// TIA Portal V15.1 export
// export: Created 2024-06-21T08:41:21.2470041Z, ExportSetting WithDefaults, DisplayName Totally Integrated Automation Portal, DisplayVersion V15.1 Update 5, DisplayName TIA Portal Openness, DisplayVersion V15.1 Update 5, DisplayName SINAMICS Startdrive Advanced, DisplayVersion V15.1, DisplayName G130, G150, S120, S150, SINAMICS MV, S210, DisplayVersion V15.1, DisplayName G110M, G120, G120C, G120D, G120P, DisplayVersion V15.1, DisplayName STEP 7 Professional, DisplayVersion V15.1 Update 5, DisplayName STEP 7 Safety, DisplayVersion V15.1, DisplayName WinCC Professional, DisplayVersion V15.1 Update 5, DisplayName SIMATIC Visualization Architect, DisplayVersion V15.1
FUNCTION_BLOCK "LVIDSQualityRequest"   // FB1220, SCL
{ S7_Optimized_Access := 'TRUE' }
VERSION : 0.1
// stored: AutoNumber false, IsIECCheckEnabled false, IsRetainMemResEnabled false, MemoryReserve 100, SetENOAutomatically False, UDAEnableTagReadback false
   VAR_INPUT
      I_TagID { ExternalAccessible := 'False'; ExternalVisible := 'False'; ExternalWritable := 'False'} : DWord;   // Tag ID
      I_BodyID { ExternalAccessible := 'False'; ExternalVisible := 'False'; ExternalWritable := 'False'} : DWord;   // Body ID
      I_CarrierID { ExternalAccessible := 'False'; ExternalVisible := 'False'; ExternalWritable := 'False'} : DWord;   // Carrier ID
      I_MixNr { ExternalAccessible := 'False'; ExternalVisible := 'False'; ExternalWritable := 'False'} : DWord;   // Mix Nr
      I_PopID { ExternalAccessible := 'False'; ExternalVisible := 'False'; ExternalWritable := 'False'} : UDInt;   // Spare Data / PopID
      I_PopIDSuffix { ExternalAccessible := 'False'; ExternalVisible := 'False'; ExternalWritable := 'False'} : Char;   // PopID suffix
      I_PopType { ExternalAccessible := 'False'; ExternalVisible := 'False'; ExternalWritable := 'False'} : UDInt;   // Pop identifier
      I_ManualModeVisible { ExternalAccessible := 'False'; ExternalVisible := 'False'; ExternalWritable := 'False'} : Bool := 0;   // 0= Hidden 1= Visible
      I_Start { ExternalAccessible := 'False'; ExternalVisible := 'False'; ExternalWritable := 'False'} : Bool;   // Start command
   END_VAR
   VAR_OUTPUT
      O_DataModeAuto { ExternalAccessible := 'False'; ExternalVisible := 'False'; ExternalWritable := 'False'} : Bool;   // Data mode - Automatic
      O_DataModeMan { ExternalAccessible := 'False'; ExternalVisible := 'False'; ExternalWritable := 'False'} : Bool;   // Data mode - Manual
      O_DataValid { ExternalAccessible := 'False'; ExternalVisible := 'False'; ExternalWritable := 'False'} : Bool;   // Data valid
      O_DataNotValid { ExternalAccessible := 'False'; ExternalVisible := 'False'; ExternalWritable := 'False'} : Bool;   // Data not valid
      O_BodyCargoStatusOk { ExternalAccessible := 'False'; ExternalVisible := 'False'; ExternalWritable := 'False'} : Bool;
      O_BodyCargoStatusNok { ExternalAccessible := 'False'; ExternalVisible := 'False'; ExternalWritable := 'False'} : Bool;
      O_Busy { ExternalAccessible := 'False'; ExternalVisible := 'False'; ExternalWritable := 'False'} : Bool;   // Busy
      O_Status { ExternalAccessible := 'False'; ExternalVisible := 'False'; ExternalWritable := 'False'} : Int;   // Status code
      O_Alarm { ExternalAccessible := 'False'; ExternalVisible := 'False'; ExternalWritable := 'False'} : Bool;   // Alarm
      O_VemData { ExternalAccessible := 'False'; ExternalVisible := 'False'; ExternalWritable := 'False'} : "VEMData";
   END_VAR
   VAR_IN_OUT
      IO_VIDS : "VIDS";   // PCS data record
      IO_Alarm : "Alarm";   // Alarm
      H_HMI : "H_HMI";
      H_LVIDSQualityRequest : "H_LVIDSQualityRequest";   // HMI - specific interface
   END_VAR
   VAR
      DataModeAuto { ExternalAccessible := 'False'; ExternalVisible := 'False'; ExternalWritable := 'False'} : Bool;
      DataModeAutoEdge { ExternalAccessible := 'False'; ExternalVisible := 'False'; ExternalWritable := 'False'} : Bool;
      DataModeAutoPls { ExternalAccessible := 'False'; ExternalVisible := 'False'; ExternalWritable := 'False'} : Bool;
      DataModeMan { ExternalAccessible := 'False'; ExternalVisible := 'False'; ExternalWritable := 'False'} : Bool;
      DataModeManEdge { ExternalAccessible := 'False'; ExternalVisible := 'False'; ExternalWritable := 'False'} : Bool;
      DataModeManPls { ExternalAccessible := 'False'; ExternalVisible := 'False'; ExternalWritable := 'False'} : Bool;
      DataModeChanged { ExternalAccessible := 'False'; ExternalVisible := 'False'; ExternalWritable := 'False'} : Bool;
      StartCmdEdgAuto { ExternalAccessible := 'False'; ExternalVisible := 'False'; ExternalWritable := 'False'} : Bool;
      StartCmdPlsAuto { ExternalAccessible := 'False'; ExternalVisible := 'False'; ExternalWritable := 'False'} : Bool;
      StartCmdPlsMan { ExternalAccessible := 'False'; ExternalVisible := 'False'; ExternalWritable := 'False'} : Bool;
      StartCmdEdgMan { ExternalAccessible := 'False'; ExternalVisible := 'False'; ExternalWritable := 'False'} : Bool;
      BeginReqPlsDataModeAuto { ExternalAccessible := 'False'; ExternalVisible := 'False'; ExternalWritable := 'False'} : Bool;
      BeginReqPlsDataModeMan { ExternalAccessible := 'False'; ExternalVisible := 'False'; ExternalWritable := 'False'} : Bool;
      Status { ExternalAccessible := 'False'; ExternalVisible := 'False'; ExternalWritable := 'False'} : Int;
      BtnModeManConfirm { ExternalAccessible := 'False'; ExternalVisible := 'False'; ExternalWritable := 'False'} : Bool;
      Alarm { ExternalAccessible := 'False'; ExternalVisible := 'False'; ExternalWritable := 'False'} : Bool;
      DataValid { ExternalAccessible := 'False'; ExternalVisible := 'False'; ExternalWritable := 'False'} : Bool;
      DataNotValid { ExternalAccessible := 'False'; ExternalVisible := 'False'; ExternalWritable := 'False'} : Bool;
      TagIDMem { ExternalAccessible := 'False'; ExternalVisible := 'False'; ExternalWritable := 'False'} : DWord;
      BodyIDMem { ExternalAccessible := 'False'; ExternalVisible := 'False'; ExternalWritable := 'False'} : DWord;
      CarrierIDMem { ExternalAccessible := 'False'; ExternalVisible := 'False'; ExternalWritable := 'False'} : DWord;
      MixNrMem { ExternalAccessible := 'False'; ExternalVisible := 'False'; ExternalWritable := 'False'} : DWord;
      PopIDMem { ExternalAccessible := 'False'; ExternalVisible := 'False'; ExternalWritable := 'False'} : UDInt;
      PopIDSuffixMem { ExternalAccessible := 'False'; ExternalVisible := 'False'; ExternalWritable := 'False'} : Char;
      PopTypeMem { ExternalAccessible := 'False'; ExternalVisible := 'False'; ExternalWritable := 'False'} : UDInt;
      BodyCargoStatusOk { ExternalAccessible := 'False'; ExternalVisible := 'False'; ExternalWritable := 'False'} : Bool;
      BodyCargoStatusNok { ExternalAccessible := 'False'; ExternalVisible := 'False'; ExternalWritable := 'False'} : Bool;
      BodyType1 { ExternalAccessible := 'False'; ExternalVisible := 'False'; ExternalWritable := 'False'} : DWord;
      VemData { ExternalAccessible := 'False'; ExternalVisible := 'False'; ExternalWritable := 'False'; S7_SetPoint := 'True'} : "VEMData";
      VemDataEmty { ExternalAccessible := 'False'; ExternalVisible := 'False'; ExternalWritable := 'False'; S7_SetPoint := 'True'} : "VEMData";
      H_btnConfirmDataModeManEnable : Word;
      H_btnConfirmDataModeManVisible : Word;
      H_txtSequenceNrEnable : Word;
      H_txtSequenceNrVisible : Word;
      H_txtSequenceNrColour : Word;
      H_txtFieldBodyType1Color : Word;
      H_txtFieldBodyType1Visible : Word;
      H_txtFieldBodyType1Enable : Word;
   END_VAR
   VAR_TEMP
      Temp_NotUsedBool : Bool;
   END_VAR
   VAR CONSTANT
      C_Command : DWord := 3041;   // Command for specific data
      OFF : Word := 2#0000000000000000;
      ENABLE : Word := 2#0000000000000001;
      VISIBLE : Word := 2#0000000000000010;
      COLOUR_GREY : Word := 2#0000000000010000;
      COLOUR_WHITE : Word := 2#0000000000100000;
      COLOUR_GREEN : Word := 2#0000000001000000;
      COLOUR_RED : Word := 2#0000000010000000;
      COLOUR_BLUE_FLASH : Word := 2#0000000100000000;
   END_VAR
BEGIN
   (******************************************************************************************  
    Changelog

       2017/06/21 AndriesHeynssens
       - Module 5005 based on the module GetSpecData build by PMo

    Description

       This module gets specific cardata from production server
       Adapt the following sections to your needs :

           IT Code 3041 Atacq

    List of authors

       Company : Volvo Cars Gent
       Name    : Patrick Moreau (PMo)
       E-mail  : patrick.moreau@volvocars.com
       Tel.    : +32 9 2503165

    ******************************************************************************************)


   (******************************************************************************)
   (* Input from HMI - Buttons                                                   *)
   (******************************************************************************)
   // FC1014
   "LDWordToBit"(I_DWord:=#H_HMI.H_CommandDW1,
                 O_0=>#BtnModeManConfirm,
                 O_1=>#Temp_NotUsedBool,
                 O_2=>#Temp_NotUsedBool,
                 O_3=>#Temp_NotUsedBool,
                 O_4=>#Temp_NotUsedBool,
                 O_5=>#Temp_NotUsedBool,
                 O_6=>#Temp_NotUsedBool,
                 O_7=>#Temp_NotUsedBool,
                 O_8=>#Temp_NotUsedBool,
                 O_9=>#Temp_NotUsedBool,
                 O_10=>#Temp_NotUsedBool,
                 O_11=>#Temp_NotUsedBool,
                 O_12=>#Temp_NotUsedBool,
                 O_13=>#Temp_NotUsedBool,
                 O_14=>#Temp_NotUsedBool,
                 O_15=>#Temp_NotUsedBool,
                 O_16=>#Temp_NotUsedBool,
                 O_17=>#Temp_NotUsedBool,
                 O_18=>#Temp_NotUsedBool,
                 O_19=>#Temp_NotUsedBool,
                 O_20=>#Temp_NotUsedBool,
                 O_21=>#Temp_NotUsedBool,
                 O_22=>#Temp_NotUsedBool,
                 O_23=>#Temp_NotUsedBool,
                 O_24=>#Temp_NotUsedBool,
                 O_25=>#Temp_NotUsedBool,
                 O_26=>#Temp_NotUsedBool,
                 O_27=>#Temp_NotUsedBool,
                 O_28=>#Temp_NotUsedBool,
                 O_29=>#Temp_NotUsedBool,
                 O_30=>#Temp_NotUsedBool,
                 O_31=>#Temp_NotUsedBool);
   #H_HMI.H_CommandDW1 := 0;

   (******************************************************************************)
   (* Data mode - Automatic                                                      *)
   (******************************************************************************)  
   //Data mode selected  - No mode, select auto
   IF (#H_LVIDSQualityRequest.H_selDataMode < 1) OR (#H_LVIDSQualityRequest.H_selDataMode > 2) OR NOT #IO_VIDS.PartPres  THEN
       #H_LVIDSQualityRequest.H_selDataMode := 1;
   END_IF;

   #DataModeAuto:=(#H_LVIDSQualityRequest.H_selDataMode=1);
   #DataModeAutoPls := #DataModeAuto AND NOT #DataModeAutoEdge;
   #DataModeAutoEdge := #DataModeAuto;

   (******************************************************************************)
   (* Data mode - Manual                                                         *)
   (******************************************************************************)
   #DataModeMan := (#H_LVIDSQualityRequest.H_selDataMode = 2);
   #DataModeManPls := #DataModeMan AND NOT #DataModeManEdge;
   #DataModeManEdge := #DataModeMan;

   (******************************************************************************)
   (* Data mode - SIMULATE                                                       *)
   (******************************************************************************)

   //Data mode changed
   #DataModeChanged := #DataModeAutoPls OR #DataModeManPls;

   (******************************************************************************************************************************)
   (* COMMUNICATION WITH IT                                                                                                      *)
   (******************************************************************************************************************************)

   (******************************************************************************)
   (* Start Pulses                                                               *)
   (******************************************************************************)
   //Start command pulse - Data mode automatic
   #StartCmdPlsAuto := #I_Start AND NOT #StartCmdEdgAuto;
   #StartCmdEdgAuto := #I_Start;

   //Start command pulse - Data mode manual
   #StartCmdPlsMan := #BtnModeManConfirm AND NOT #StartCmdEdgMan;    
   #StartCmdEdgMan := #BtnModeManConfirm;

   (******************************************************************************)
   (* Begin request                                                              *)
   (******************************************************************************)

   //Begin request
   #BeginReqPlsDataModeAuto := (#StartCmdPlsAuto AND #DataModeAuto);
   #BeginReqPlsDataModeMan := (#StartCmdPlsMan AND #DataModeMan);

   #IO_VIDS.GetSpecData.BeginReq := #BeginReqPlsDataModeAuto OR #BeginReqPlsDataModeMan;

   IF  #IO_VIDS.GetSpecData.BeginReq THEN
       #Status := 0;
       #TagIDMem := #I_TagID;
       #BodyIDMem := #I_BodyID;
       #CarrierIDMem := #I_CarrierID;
       #MixNrMem := #I_MixNr;
       #PopIDMem := #I_PopID;
       #PopIDSuffixMem := #I_PopIDSuffix;
       #PopTypeMem := #I_PopType;
   END_IF;

   (******************************************************************************)
   (* OkBegin / Begin / Running                                                  *)
   (******************************************************************************)
   //OkBegin
   IF  #IO_VIDS.GetSpecData.OkBegin THEN
       #DataValid := False;
       #DataNotValid := False;
       #IO_VIDS.VEMData.FunctionCode := 0; //>>> MOET "0" ZIJN >>> DECODE YOUR DATA HERE!
       #IO_VIDS.VEMData.CommandCode := #C_Command; //>>> DECODE YOUR DATA HERE!
       #IO_VIDS.VEMData.Identification:= #TagIDMem; //>>> DECODE YOUR DATA HERE!
       #IO_VIDS.VEMData.BodyID:= #BodyIDMem; //>>> DECODE YOUR DATA HERE!
       #IO_VIDS.VEMData.CarrierID := #CarrierIDMem; //>>> DECODE YOUR DATA HERE!
       #IO_VIDS.VEMData.MixNumber := #MixNrMem; //>>> DECODE YOUR DATA HERE!
       #IO_VIDS.VEMData.PopID := #PopIDMem; //>>> DECODE YOUR DATA HERE!
       #IO_VIDS.VEMData.PopIDSuffix := #PopIDSuffixMem; //>>> DECODE YOUR DATA HERE!
       #IO_VIDS.VEMData.PopType := #PopTypeMem; //>>> DECODE YOUR DATA HERE!
   END_IF;

   //Begin
   #IO_VIDS.GetSpecData.Begin := #IO_VIDS.GetSpecData.OkBegin;

   //Running
   IF #IO_VIDS.GetSpecData.Running THEN
       #Status := #IO_VIDS.GetSpecData.Status;
   END_IF;

   (******************************************************************************)
   (* Finish                                                                     *)
   (******************************************************************************)
   IF #IO_VIDS.GetSpecData.Finished THEN
       #Status := #IO_VIDS.GetSpecData.Status;

       IF #Status = 1 THEN
           #BodyType1 := #IO_VIDS.VEMData.BodyType1; //>>> DECODE YOUR DATA HERE! 
           #VemData := #IO_VIDS.VEMData; //>>> DECODE YOUR DATA HERE! 
           #DataValid := TRUE;
       ELSE
               #DataNotValid := TRUE;
       END_IF;

   END_IF;

   (******************************************************************************************************************************)
   (* EINDE COMMUNICATION WITH IT                                                                                                *)
   (******************************************************************************************************************************)

   (******************************************************************************)
   (* Clear data                                                                 *)
   (******************************************************************************)
   IF #IO_VIDS.GetSpecData.BeginReq OR #DataModeChanged OR NOT #IO_VIDS.PartPres THEN
       #DataValid := False;
       #DataNotValid := False;
       #Status := 0;
       #BodyType1 := 0;//>>> DECODE YOUR DATA HERE! 
       #VemData := #VemDataEmty;//>>> DECODE YOUR DATA HERE! 

   END_IF;

   IF NOT #IO_VIDS.PartPres THEN
       #TagIDMem := 0;//>>> DECODE YOUR DATA HERE!
       #BodyIDMem := 0;//>>> DECODE YOUR DATA HERE!
       #CarrierIDMem := 0;//>>> DECODE YOUR DATA HERE!
       #MixNrMem := 0;//>>> DECODE YOUR DATA HERE!
       #PopIDMem := 0;//>>> DECODE YOUR DATA HERE!
       #PopIDSuffixMem := ' ';//>>> DECODE YOUR DATA HERE!
       #PopTypeMem := 0;//>>> DECODE YOUR DATA HERE!
   END_IF;

   (******************************************************************************)
   (* Alarm = status <0                                                          *)
   (******************************************************************************)
   IF #Status < 0 THEN
       #Alarm := TRUE;
   ELSE
       #Alarm := false;
   END_IF;

   "LAlarmSummary"(I_AlarmA := FALSE,
                   I_AlarmB := FALSE,
                   I_AlarmC := #Alarm,
                   I_AlarmD := FALSE,
                   I_AlarmABCondition := FALSE,
                   IO_Alarm := #IO_Alarm,
                   C_UpperLevelHW := "FALSE",
                   C_UpperLevelSafety := "FALSE",
                   C_Safety := "FALSE",
                   C_Mechanic := "FALSE",
                   C_Transport := "FALSE",
                   C_Feature1 := "FALSE",
                   C_Feature2 := "FALSE",
                   C_Feature3 := "FALSE");

   (******************************************************************************)
   (* Calculation BodyCargoStatus OK - NOK                                       *)
   (******************************************************************************)

   IF #VemData.BodyCargoStatus.%X0 = true THEN
       #BodyCargoStatusOk := TRUE;
   ELSE
       #BodyCargoStatusOk := FALSE;
   END_IF;

   IF #VemData.BodyCargoStatus.%X1 = true THEN
       #BodyCargoStatusNok := TRUE;
   ELSE
       #BodyCargoStatusNok := FALSE;
   END_IF;

   (******************************************************************************)
   (* Outputs                                                                    *)
   (******************************************************************************)
   #O_DataModeAuto := #DataModeAuto;
   #O_DataModeMan := #DataModeMan;
   #O_DataValid := #DataValid;
   #O_DataNotValid := #DataNotValid;
   #O_Alarm := #Alarm;
   #O_Status := #Status;
   #O_Busy := #IO_VIDS.GetSpecData.Running;
   #O_VemData := #VemData;                         //>>> DECODE YOUR DATA HERE!
   #O_BodyCargoStatusOk := #BodyCargoStatusOk;     //>>> DECODE YOUR DATA HERE!
   #O_BodyCargoStatusNok := #BodyCargoStatusNok;   //>>> DECODE YOUR DATA HERE!

   (******************************************************************************************************************************)
   (* Animations                                                                                                                 *)
   (******************************************************************************************************************************)

   (******************************************************************************)
   (* Status To HMI word                                                         *)
   (******************************************************************************)
   "LBitToDword"(I_0:=#IO_VIDS.PartPres,
                 I_1:=#DataValid,
                 I_2:=#DataNotValid,
                 I_3:=#Alarm,
                 I_4:=#I_Start,
                 I_5:=#H_LVIDSQualityRequest.H_selDataMode = 3,
                 I_6:=FALSE,
                 I_7:=FALSE,
                 I_8:=FALSE,
                 I_9:=FALSE,
                 I_10:=FALSE,
                 I_11:=FALSE,
                 I_12:=FALSE,
                 I_13:=FALSE,
                 I_14:=FALSE,
                 I_15:=FALSE,
                 I_16:=FALSE,
                 I_17:=FALSE,
                 I_18:=FALSE,
                 I_19:=FALSE,
                 I_20:=FALSE,
                 I_21:=FALSE,
                 I_22:=FALSE,
                 I_23:=FALSE,
                 I_24:=FALSE,
                 I_25:=FALSE,
                 I_26:=FALSE,
                 I_27:=FALSE,
                 I_28:=FALSE,
                 I_29:=FALSE,
                 I_30:=FALSE,
                 I_31:=FALSE,
                 O_DWord=>#H_LVIDSQualityRequest.H_Anim);

   (******************************************************************************)
   (* Status To HMI word - IAnim                                                 *)
   (******************************************************************************)
   //*** Machine #Status - Indication *** TO HMI - Icon animation
   "LIAnimDWord"(I_SetPos:=FALSE,
                 I_ResetPos:=FALSE,
                 I_Active:=#Status=2,
                 I_Visible:=FALSE,
                 I_OutOfUse:=FALSE,
                 I_IntlkSet:=FALSE,
                 I_IntlkReset:=FALSE,
                 I_IntlkSetAlm:=FALSE,
                 I_IntlkResetAlm:=FALSE,
                 I_ManualMode:=FALSE,
                 I_FncSelInHMI:=FALSE,
                 I_AnySelected:=FALSE,
                 I_AlarmA:=FALSE,
                 I_AlarmB:=FALSE,
                 I_AlarmC:=#DataNotValid,
                 I_AlarmD:=FALSE,
                 I_SafetyOk:=FALSE,
                 I_Service:=TRUE,
                 I_Spare1:=FALSE,
                 I_Spare2:=FALSE,
                 I_Spare3:=FALSE,
                 I_Spare4:=FALSE,
                 I_Spare5:=FALSE,
                 I_Spare6:=FALSE,
                 I_Spare7:=FALSE,
                 I_Spare8:=FALSE,
                 I_Spare9:=FALSE,
                 I_Spare10:=FALSE,
                 I_Spare11:=FALSE,
                 I_Spare12:=FALSE,
                 I_Spare13:=FALSE,
                 I_Spare14:=FALSE,
                 H_IAnim=>#H_HMI.H_IAnim);

   (******************************************************************************)
   (* Copy Txt info to HMI                                                       *)
   (******************************************************************************)
   #H_LVIDSQualityRequest.H_txtStatusIT := #Status;
   #H_LVIDSQualityRequest.H_txtBodyCargoStatus := #VemData.BodyCargoStatus;
   #H_LVIDSQualityRequest.H_txtRouting := #VemData.Routing;
   #H_LVIDSQualityRequest.H_txtPopType := #VemData.PopType;
   #H_LVIDSQualityRequest.H_txtPopId := #VemData.PopID;
   #H_LVIDSQualityRequest.H_txtPopIdSuffix := #VemData.PopIDSuffix;

   #H_LVIDSQualityRequest.H_txtInTagID := #TagIDMem;
   #H_LVIDSQualityRequest.H_txtInBodyID := #BodyIDMem;
   #H_LVIDSQualityRequest.H_txtInCarrierID := #CarrierIDMem;
   #H_LVIDSQualityRequest.H_txtInMixNr := #MixNrMem;
   #H_LVIDSQualityRequest.H_txtInPopId := #PopIDMem;
   #H_LVIDSQualityRequest.H_txtInPopIdSuffix := #PopIDSuffixMem;
   #H_LVIDSQualityRequest.H_txtInPopType := #PopTypeMem;

   #H_LVIDSQualityRequest.H_txtCommandCodeRcvd := #IO_VIDS.CmdCodeRcvd;
   #H_LVIDSQualityRequest.H_txtCommandCodeSent := #IO_VIDS.CmdCodeSent;

   (******************************************************************************)
   (* Animation BUTTONS                                                          *)
   (******************************************************************************)
   //Data mode manual - <Confirm> button
   IF #I_ManualModeVisible AND #DataModeMan THEN
       #H_btnConfirmDataModeManVisible := #VISIBLE;
       #H_btnConfirmDataModeManEnable := #ENABLE;
   ELSE
       #H_btnConfirmDataModeManVisible := #OFF;
       #H_btnConfirmDataModeManEnable := #OFF;
   END_IF;

   #H_LVIDSQualityRequest.H_btnConfirmDataModeManAnim := #H_btnConfirmDataModeManEnable OR #H_btnConfirmDataModeManVisible;
END_FUNCTION_BLOCK
